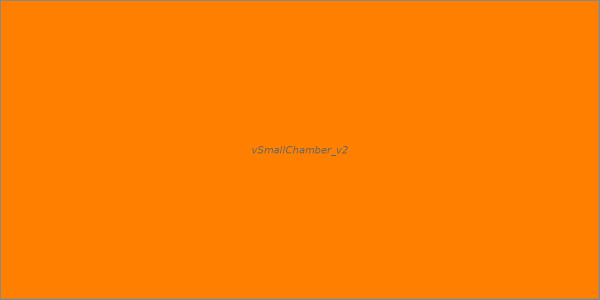
VISUALIZATION vStatusScreen_v2  // 600x300
VAR_IN_OUT
	arChamber :  fbChamber;
	arParams :    stParamsChamber;
	arControl :    stControl;
END_VAR
    Frame (0,0 600x300)
        shows vSmallChamber_v2(stParams := arParams, fbChamber := arChamber, stControl := arControl)
END_VISUALIZATION

(* stored: Version 1.1.0.1, ProductVersion 3.1.4024.12
   Visu vStatusScreen_v2: Id {4fd026e6-26e2-455a-9971-e3a064ef64f8} *)
